// TIA Portal V17 export
// export: Created 2024-09-02T12:50:26.3291542Z, ExportSetting WithDefaults, DisplayName Totally Integrated Automation Portal, DisplayVersion V17, DisplayName TIA Portal Openness, DisplayVersion V17, DisplayName TIA Portal Version Control Interface, DisplayVersion V17, DisplayName STEP 7 Professional, DisplayVersion V17, DisplayName STEP 7 Safety, DisplayVersion V17, DisplayName WinCC Professional, DisplayVersion V17
TYPE "TypeOperatingModesGlobal"
// stored: IsFailsafeCompliant false
   STRUCT
      machine_on : Bool;   // Anlage einschalten / Switch on the system
      machine_ready : Bool;   // Anlage hochgefahren / Plant started up
      machine_startup_active : Bool;   // Anlagenochlauf aktiv / System run-up active
      machine_startup_fp_quit_01 : Bool;   // Anlagenochlauf: Flanke Quitt. 01 / System run-up: Edge Acknowledge 01
      machine_startup_fp_quit_02 : Bool;   // Anlagenochlauf: Flanke Quitt. 02 / System run-up: Edge Acknowledge 02
      machine_startup_fp_quit_03 : Bool;   // Anlagenochlauf: Flanke Quitt. 03 / System run-up: Edge Acknowledgement 03
      machine_startup_hm_quit_01 : Bool;   // Anlagenochlauf:HM Quitt. 01 / System run-up:HM Receipt. 01
      machine_startup_hm_quit_02 : Bool;   // Anlagenochlauf:HM Quitt. 02 / System run-up:HM Quitt. 02
      machine_startup_hm_quit_03 : Bool;   // Anlagenochlauf:HM Quitt. 03 / System run-up:HM Quitt. 03
      para_machine_startupTime : Time;   // Parameter: Anlagenhochlaufzeit / Parameters: system ramp-up time
      rest_machine_startuplTime : Time;   // Rest Anlagenhochlaufzeit / Rest of investment ramp-up time
      profinetfault : Bool;   // Profinetstörung / Profinet disorder
      tln_profinetfault : Int;   // TLN Profinetstörung / TLN Profinet disturbance
      StartupTime { S7_SetPoint := 'True'} : TP_TIME;   // Timer: Anlagenhochlaufzeit / Timer: System ramp-up time
      ErrorTimeTempSS { S7_SetPoint := 'True'} : TON_TIME;   // Temperaturfehler Schaltschrank / Temperature error control cabinet
      "Time" { ExternalWritable := 'False'; S7_SetPoint := 'True'} : Array[1..9] of IEC_TIMER;   // IEC Time
      hm_ErrorTempSS : Array[1..8] of Bool;   // HM Temperaturfehler Schaltschrank / HM Temperature error Switch cabinet
   END_STRUCT;
END_TYPE
